% RSLogix 500 project PROJECT2.RSS, saved by version 8.30.00.16 %
PROJECT "PROJECT2"    % processor: Bul.1763 MicroLogix 1100 Series B %

PROGRAM FILES
  LAD 2 "MAIN"  3 rungs
  LAD 3 "DI/DO"  8 rungs
  LAD 4 "CONTROL"  4 rungs

DATA FILES
  O0 OUTPUT  5 elements
  I1 INPUT  7 elements
  S2 STATUS  66 elements
  B3 BINARY  1 elements
  T4 TIMER  1 elements
  C5 COUNTER  1 elements
  R6 CONTROL  1 elements
  N7 INTEGER  1 elements
  F8 FLOAT  1 elements

LADDER 2 "MAIN"
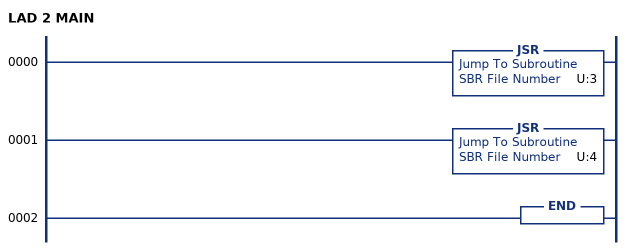
% Rung: 0 %
SOR JSR U:3 EOR
% Rung: 1 %
SOR JSR U:4 EOR
% Rung: 2 %
SOR END EOR

LADDER 3 "DI/DO"
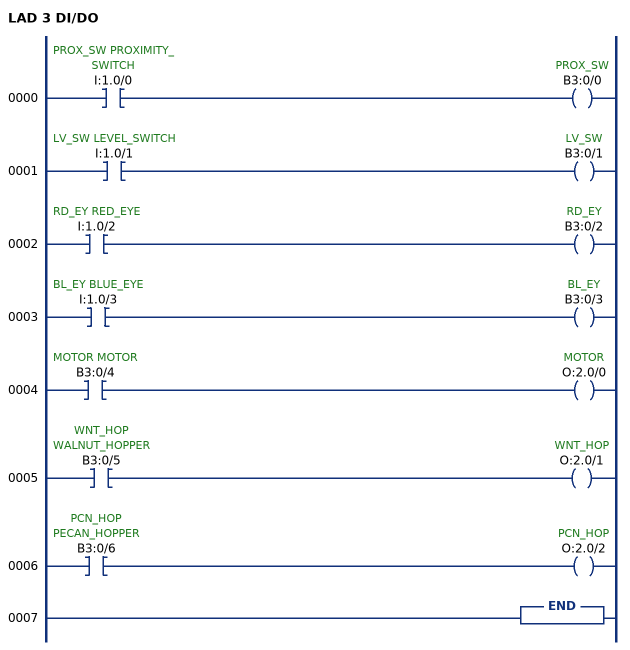
% Rung: 0 %
SOR XIC I:1.0/0 OTE B3:0/0 EOR
%   I:1.0/0  PROXIMITY_SWITCH  "PROX_SW" %
%   B3:0/0  "PROX_SW" %
% Rung: 1 %
SOR XIC I:1.0/1 OTE B3:0/1 EOR
%   I:1.0/1  LEVEL_SWITCH  "LV_SW" %
%   B3:0/1  "LV_SW" %
% Rung: 2 %
SOR XIC I:1.0/2 OTE B3:0/2 EOR
%   I:1.0/2  RED_EYE  "RD_EY" %
%   B3:0/2  "RD_EY" %
% Rung: 3 %
SOR XIC I:1.0/3 OTE B3:0/3 EOR
%   I:1.0/3  BLUE_EYE  "BL_EY" %
%   B3:0/3  "BL_EY" %
% Rung: 4 %
SOR XIC B3:0/4 OTE O:2.0/0 EOR
%   B3:0/4  MOTOR  "MOTOR" %
%   O:2.0/0  "MOTOR" %
% Rung: 5 %
SOR XIC B3:0/5 OTE O:2.0/1 EOR
%   B3:0/5  WALNUT_HOPPER  "WNT_HOP" %
%   O:2.0/1  "WNT_HOP" %
% Rung: 6 %
SOR XIC B3:0/6 OTE O:2.0/2 EOR
%   B3:0/6  PECAN_HOPPER  "PCN_HOP" %
%   O:2.0/2  "PCN_HOP" %
% Rung: 7 %
SOR END EOR

LADDER 4 "CONTROL"
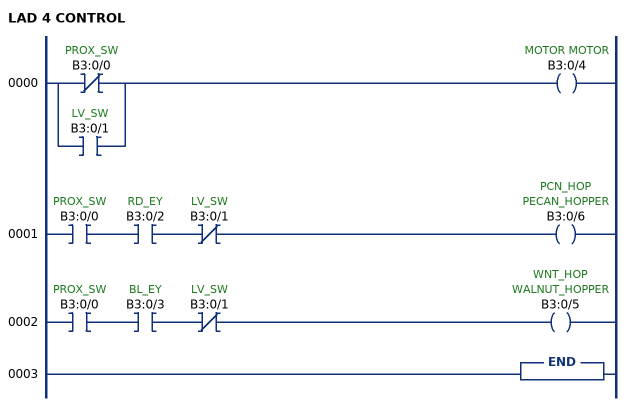
% Rung: 0 %
SOR BST XIO B3:0/0 NXB XIC B3:0/1 BND OTE B3:0/4 EOR
%   B3:0/0  "PROX_SW" %
%   B3:0/1  "LV_SW" %
%   B3:0/4  MOTOR  "MOTOR" %
% Rung: 1 %
SOR XIC B3:0/0 XIC B3:0/2 XIO B3:0/1 OTE B3:0/6 EOR
%   B3:0/0  "PROX_SW" %
%   B3:0/2  "RD_EY" %
%   B3:0/1  "LV_SW" %
%   B3:0/6  PECAN_HOPPER  "PCN_HOP" %
% Rung: 2 %
SOR XIC B3:0/0 XIC B3:0/3 XIO B3:0/1 OTE B3:0/5 EOR
%   B3:0/0  "PROX_SW" %
%   B3:0/3  "BL_EY" %
%   B3:0/1  "LV_SW" %
%   B3:0/5  WALNUT_HOPPER  "WNT_HOP" %
% Rung: 3 %
SOR END EOR
